PROGRAM prg_Millis
VAR
	tpMillis : TP;
	bPuls	AT		%Q*		:BOOL;
END_VAR

tpMillis(IN := NOT tpMillis.Q, PT := T#1S);
bPuls := NOT(tpMillis.Q);

//Als je dit in 1 regel wilt moet je gewoon bPuls bij de Q van tpmillis zetten

END_PROGRAM

(* stored: Version 1.1.0.1, ProductVersion 3.1.4024.15
   POU prg_Millis: Id {dd5a5dd1-f5f8-4920-a311-12fff34722f3}, SpecialFunc None *)
